// TIA Portal V18 export
// export: Created 2026-01-09T11:31:53.9604864Z, ExportSetting WithDefaults, DisplayName Totally Integrated Automation Portal, DisplayVersion V18 Update 5, DisplayName TIA Portal Openness, DisplayVersion V18 Update 5, DisplayName TIA Portal Teamcenter Gateway, DisplayVersion V18, DisplayName TIA Portal Version Control Interface, DisplayVersion V18, DisplayName SINAMICS Startdrive Advanced, DisplayVersion V18 SP2 Update 1, DisplayName SINAMICS Startdrive G110M, G120, G120C, G120D, G120P, G115D, DisplayVersion V18 SP2 Update 1, DisplayName SINAMICS Startdrive G130, G150, S120, S150, SINAMICS MV, S210, G220, S200, DisplayVersion V18 SP2 Update 1, DisplayName STEP 7 Professional, DisplayVersion V18 Update 5, DisplayName STEP 7 Safety, DisplayVersion V18, DisplayName WinCC Professional, DisplayVersion V18 Update 5
TagTable "NG"
  PalletNGData_LoadingNGPallet_NG_1_1 : Bool  (PLC tag PalletNGData.LoadingNGPallet.NG_1_1, CPU S71500-2PN_TP700, 100 ms)
  PalletNGData_LoadingNGPallet_NG_1_2 : Bool  (PLC tag PalletNGData.LoadingNGPallet.NG_1_2, CPU S71500-2PN_TP700, 100 ms)
  PalletNGData_LoadingNGPallet_NG_1_3 : Bool  (PLC tag PalletNGData.LoadingNGPallet.NG_1_3, CPU S71500-2PN_TP700, 100 ms)
  PalletNGData_LoadingNGPallet_NG_1_4 : Bool  (PLC tag PalletNGData.LoadingNGPallet.NG_1_4, CPU S71500-2PN_TP700, 100 ms)
  PalletNGData_LoadingNGPallet_NG_1_5 : Bool  (PLC tag PalletNGData.LoadingNGPallet.NG_1_5, CPU S71500-2PN_TP700, 100 ms)
  PalletNGData_LoadingNGPallet_NG_2_1 : Bool  (PLC tag PalletNGData.LoadingNGPallet.NG_2_1, CPU S71500-2PN_TP700, 100 ms)
  PalletNGData_LoadingNGPallet_NG_2_2 : Bool  (PLC tag PalletNGData.LoadingNGPallet.NG_2_2, CPU S71500-2PN_TP700, 100 ms)
  PalletNGData_LoadingNGPallet_NG_2_3 : Bool  (PLC tag PalletNGData.LoadingNGPallet.NG_2_3, CPU S71500-2PN_TP700, 100 ms)
  PalletNGData_LoadingNGPallet_NG_2_4 : Bool  (PLC tag PalletNGData.LoadingNGPallet.NG_2_4, CPU S71500-2PN_TP700, 100 ms)
  PalletNGData_LoadingNGPallet_NG_2_5 : Bool  (PLC tag PalletNGData.LoadingNGPallet.NG_2_5, CPU S71500-2PN_TP700, 100 ms)
  PalletNGData_LoadingNGPallet_NG_3_1 : Bool  (PLC tag PalletNGData.LoadingNGPallet.NG_3_1, CPU S71500-2PN_TP700, 100 ms)
  PalletNGData_LoadingNGPallet_NG_3_2 : Bool  (PLC tag PalletNGData.LoadingNGPallet.NG_3_2, CPU S71500-2PN_TP700, 100 ms)
  PalletNGData_LoadingNGPallet_NG_3_3 : Bool  (PLC tag PalletNGData.LoadingNGPallet.NG_3_3, CPU S71500-2PN_TP700, 100 ms)
  PalletNGData_LoadingNGPallet_NG_3_4 : Bool  (PLC tag PalletNGData.LoadingNGPallet.NG_3_4, CPU S71500-2PN_TP700, 100 ms)
  PalletNGData_LoadingNGPallet_NG_3_5 : Bool  (PLC tag PalletNGData.LoadingNGPallet.NG_3_5, CPU S71500-2PN_TP700, 100 ms)
  PalletNGData_LoadingNGPallet_Status_1 : Int  (PLC tag PalletNGData.LoadingNGPallet.Status_1, CPU S71500-2PN_TP700, 100 ms)
  PalletNGData_LoadingNGPallet_Status_2 : Int  (PLC tag PalletNGData.LoadingNGPallet.Status_2, CPU S71500-2PN_TP700, 100 ms)
  PalletNGData_LoadingNGPallet_Status_3 : Int  (PLC tag PalletNGData.LoadingNGPallet.Status_3, CPU S71500-2PN_TP700, 100 ms)
  PalletNGData_LoadingNGPallet_Ready_1 : Bool  (PLC tag PalletNGData.LoadingNGPallet.Ready_1, CPU S71500-2PN_TP700, 100 ms)
  PalletNGData_LoadingNGPallet_Ready_2 : Bool  (PLC tag PalletNGData.LoadingNGPallet.Ready_2, CPU S71500-2PN_TP700, 100 ms)
  PalletNGData_LoadingNGPallet_Ready_3 : Bool  (PLC tag PalletNGData.LoadingNGPallet.Ready_3, CPU S71500-2PN_TP700, 100 ms)
  PalletNGData_LoadingNGPallet_Interlock_1 : Array [0..9] of Bool  (PLC tag PalletNGData.LoadingNGPallet.Interlock_1, CPU S71500-2PN_TP700, 1 s)
    TagArrayMember "[0]"
    TagArrayMember "[1]"
    TagArrayMember "[2]"
    TagArrayMember "[3]"
    TagArrayMember "[4]"
    TagArrayMember "[5]"
    TagArrayMember "[6]"
    TagArrayMember "[7]"
    TagArrayMember "[8]"
    TagArrayMember "[9]"
  PalletNGData_LoadingNGPallet_Interlock_2 : Array [0..9] of Bool  (PLC tag PalletNGData.LoadingNGPallet.Interlock_2, CPU S71500-2PN_TP700, 1 s)
    TagArrayMember "[0]"
    TagArrayMember "[1]"
    TagArrayMember "[2]"
    TagArrayMember "[3]"
    TagArrayMember "[4]"
    TagArrayMember "[5]"
    TagArrayMember "[6]"
    TagArrayMember "[7]"
    TagArrayMember "[8]"
    TagArrayMember "[9]"
  PalletNGData_LoadingNGPallet_Interlock_3 : Array [0..9] of Bool  (PLC tag PalletNGData.LoadingNGPallet.Interlock_3, CPU S71500-2PN_TP700, 1 s)
    TagArrayMember "[0]"
    TagArrayMember "[1]"
    TagArrayMember "[2]"
    TagArrayMember "[3]"
    TagArrayMember "[4]"
    TagArrayMember "[5]"
    TagArrayMember "[6]"
    TagArrayMember "[7]"
    TagArrayMember "[8]"
    TagArrayMember "[9]"
  PalletNGData_LoadingNGPallet_LockStatus : Int  (PLC tag PalletNGData.LoadingNGPallet.LockStatus, CPU S71500-2PN_TP700, 1 s)
  PalletNGData_UnLoadingNGPallet_NG_1_1 : Bool  (PLC tag PalletNGData.UnLoadingNGPallet.NG_1_1, CPU S71500-2PN_TP700, 100 ms)
  PalletNGData_UnLoadingNGPallet_NG_1_2 : Bool  (PLC tag PalletNGData.UnLoadingNGPallet.NG_1_2, CPU S71500-2PN_TP700, 100 ms)
  PalletNGData_UnLoadingNGPallet_NG_1_3 : Bool  (PLC tag PalletNGData.UnLoadingNGPallet.NG_1_3, CPU S71500-2PN_TP700, 100 ms)
  PalletNGData_UnLoadingNGPallet_NG_1_4 : Bool  (PLC tag PalletNGData.UnLoadingNGPallet.NG_1_4, CPU S71500-2PN_TP700, 100 ms)
  PalletNGData_UnLoadingNGPallet_NG_1_5 : Bool  (PLC tag PalletNGData.UnLoadingNGPallet.NG_1_5, CPU S71500-2PN_TP700, 100 ms)
  PalletNGData_UnLoadingNGPallet_NG_2_1 : Bool  (PLC tag PalletNGData.UnLoadingNGPallet.NG_2_1, CPU S71500-2PN_TP700, 100 ms)
  PalletNGData_UnLoadingNGPallet_NG_2_2 : Bool  (PLC tag PalletNGData.UnLoadingNGPallet.NG_2_2, CPU S71500-2PN_TP700, 100 ms)
  PalletNGData_UnLoadingNGPallet_NG_2_3 : Bool  (PLC tag PalletNGData.UnLoadingNGPallet.NG_2_3, CPU S71500-2PN_TP700, 100 ms)
  PalletNGData_UnLoadingNGPallet_NG_2_4 : Bool  (PLC tag PalletNGData.UnLoadingNGPallet.NG_2_4, CPU S71500-2PN_TP700, 100 ms)
  PalletNGData_UnLoadingNGPallet_NG_2_5 : Bool  (PLC tag PalletNGData.UnLoadingNGPallet.NG_2_5, CPU S71500-2PN_TP700, 100 ms)
  PalletNGData_UnLoadingNGPallet_NG_3_1 : Bool  (PLC tag PalletNGData.UnLoadingNGPallet.NG_3_1, CPU S71500-2PN_TP700, 100 ms)
  PalletNGData_UnLoadingNGPallet_NG_3_2 : Bool  (PLC tag PalletNGData.UnLoadingNGPallet.NG_3_2, CPU S71500-2PN_TP700, 100 ms)
  PalletNGData_UnLoadingNGPallet_NG_3_3 : Bool  (PLC tag PalletNGData.UnLoadingNGPallet.NG_3_3, CPU S71500-2PN_TP700, 100 ms)
  PalletNGData_UnLoadingNGPallet_NG_3_4 : Bool  (PLC tag PalletNGData.UnLoadingNGPallet.NG_3_4, CPU S71500-2PN_TP700, 100 ms)
  PalletNGData_UnLoadingNGPallet_NG_3_5 : Bool  (PLC tag PalletNGData.UnLoadingNGPallet.NG_3_5, CPU S71500-2PN_TP700, 100 ms)
  PalletNGData_UnLoadingNGPallet_Status_1 : Int  (PLC tag PalletNGData.UnLoadingNGPallet.Status_1, CPU S71500-2PN_TP700, 100 ms)
  PalletNGData_UnLoadingNGPallet_Status_2 : Int  (PLC tag PalletNGData.UnLoadingNGPallet.Status_2, CPU S71500-2PN_TP700, 100 ms)
  PalletNGData_UnLoadingNGPallet_Status_3 : Int  (PLC tag PalletNGData.UnLoadingNGPallet.Status_3, CPU S71500-2PN_TP700, 100 ms)
  PalletNGData_UnLoadingNGPallet_Ready_1 : Bool  (PLC tag PalletNGData.UnLoadingNGPallet.Ready_1, CPU S71500-2PN_TP700, 100 ms)
  PalletNGData_UnLoadingNGPallet_Ready_2 : Bool  (PLC tag PalletNGData.UnLoadingNGPallet.Ready_2, CPU S71500-2PN_TP700, 100 ms)
  PalletNGData_UnLoadingNGPallet_Ready_3 : Bool  (PLC tag PalletNGData.UnLoadingNGPallet.Ready_3, CPU S71500-2PN_TP700, 100 ms)
  PalletNGData_UnLoadingNGPallet_Interlock_1 : Array [0..9] of Bool  (PLC tag PalletNGData.UnLoadingNGPallet.Interlock_1, CPU S71500-2PN_TP700, 1 s)
    TagArrayMember "[0]"
    TagArrayMember "[1]"
    TagArrayMember "[2]"
    TagArrayMember "[3]"
    TagArrayMember "[4]"
    TagArrayMember "[5]"
    TagArrayMember "[6]"
    TagArrayMember "[7]"
    TagArrayMember "[8]"
    TagArrayMember "[9]"
  PalletNGData_UnLoadingNGPallet_Interlock_2 : Array [0..9] of Bool  (PLC tag PalletNGData.UnLoadingNGPallet.Interlock_2, CPU S71500-2PN_TP700, 1 s)
    TagArrayMember "[0]"
    TagArrayMember "[1]"
    TagArrayMember "[2]"
    TagArrayMember "[3]"
    TagArrayMember "[4]"
    TagArrayMember "[5]"
    TagArrayMember "[6]"
    TagArrayMember "[7]"
    TagArrayMember "[8]"
    TagArrayMember "[9]"
  PalletNGData_UnLoadingNGPallet_Interlock_3 : Array [0..9] of Bool  (PLC tag PalletNGData.UnLoadingNGPallet.Interlock_3, CPU S71500-2PN_TP700, 1 s)
    TagArrayMember "[0]"
    TagArrayMember "[1]"
    TagArrayMember "[2]"
    TagArrayMember "[3]"
    TagArrayMember "[4]"
    TagArrayMember "[5]"
    TagArrayMember "[6]"
    TagArrayMember "[7]"
    TagArrayMember "[8]"
    TagArrayMember "[9]"
  PalletNGData_UnLoadingNGPallet_LockStatus : Int  (PLC tag PalletNGData.UnLoadingNGPallet.LockStatus, CPU S71500-2PN_TP700, 1 s)
